Staubli VAL3: JudgePeak.pgx

program JudgePeak()
begin
  //判断路径中的转折点
  //
end
